RoboDK station: Deburring.rdk

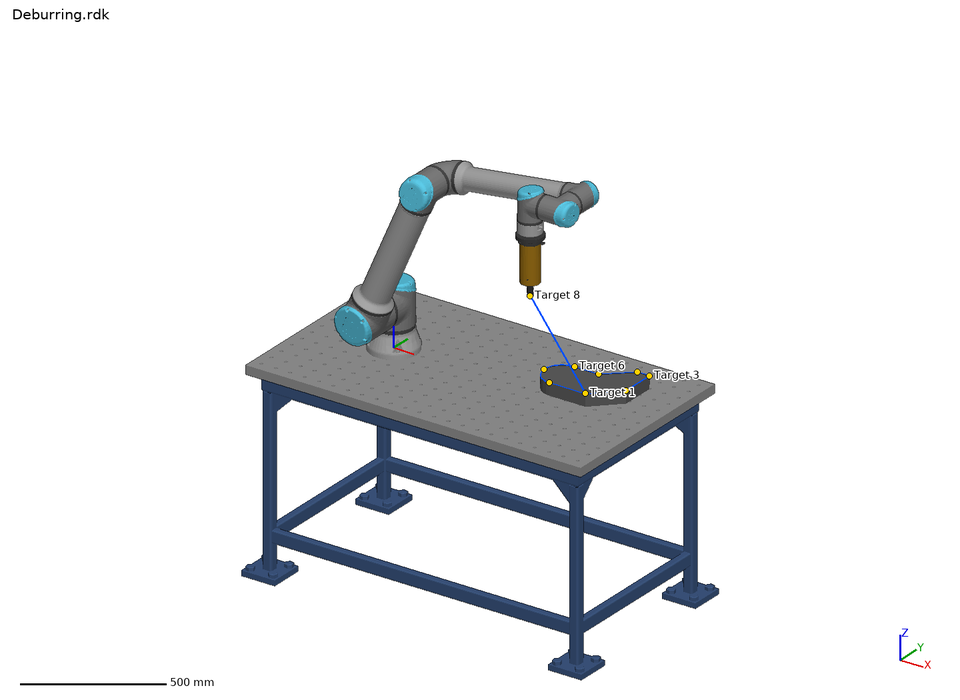
[picture v0: the station drawn from its stored meshes, robots at their saved joint values, targets as dots, program paths as lines]
Station Deburring (saved by RoboDK 5.9.2). Poses are relative to the parent item; angles as X-Y-Z fixed-axis rotations.
  - frame UR10e Base at (0, 0, 0) mm
    - robot UR10e: 6 axes, payload 10 kg, reach 1300 mm, repeatability 0.05 mm, weight 28.9 kg
        modified DH rows (alpha deg, a mm, theta deg, d mm): 0, 0, 0, 180.7; 90, 0, 180, 0; 0, 612.6, 0, 0; 0, 571.335, 0, 174.15; -90, 0, 0, 119.85; 90, 0, 180, 116.55
        joint limits [-360, -360, -360, -360, -360, -360] to [360, 360, 360, 360, 360, 360]; home [0, -90, -90, 0, 90, 0]; saved at [0, -113.502, -59.226, 82.728, 270, 180]
      - tool ATI 9150-CDB-8-11-000 Deburring Tool (Spring), TCP at (0, 0, 236.5) mm, size 103 x 103 x 235.8 mm
    - target Target 1 (Cartesian target) at (800, 0, 50) mm, rotated rx -179.28 ry 0 rz 0 deg; joints [12.276, -111.55, -108.716, -49.582, 90.702, 282.276] of UR10e
    - target Target 2 (Cartesian target) at (900, 100, 50) mm, rotated rx -179.28 ry 0 rz 0 deg; joints [17.172, -119.673, -95.84, -54.275, 90.686, 287.174] of UR10e
    - target Target 3 (Cartesian target) at (900, 240, 50) mm, rotated rx -179.28 ry 0 rz 0 deg; joints [25.472, -121.667, -92.542, -55.482, 90.648, 295.474] of UR10e
    - target Target 4 (Cartesian target) at (850, 240, 50) mm, rotated rx -179.28 ry 0 rz 0 deg; joints [26.894, -117.902, -98.773, -53.001, 90.64, 296.896] of UR10e
    - target Target 5 (Cartesian target) at (750, 150, 50) mm, rotated rx -179.28 ry 0 rz 0 deg; joints [24.18, -108.782, -112.877, -48.046, 90.655, 294.181] of UR10e
    - target Target 6 (Cartesian target) at (650, 150, 50) mm, rotated rx -179.28 ry 0 rz 0 deg; joints [27.801, -100.961, -123.659, -45.046, 90.635, 297.803] of UR10e
    - target Target 7 (Cartesian target) at (650, 0, 50) mm, rotated rx -179.28 ry 0 rz 0 deg; joints [15.174, -99.587, -125.359, -44.866, 90.693, 285.175] of UR10e
    - target Target 8 (Cartesian target) at (691.19, -174.15, 461.75) mm, rotated rx -180 ry 0 rz -90 deg; joints [0, -90, -90, -90, 90, 0] of UR10e
    - target Target 9 (Cartesian target) at (575, 75, 50) mm, rotated rx -179.28 ry 0 rz 0 deg; joints [24.517, -93.386, -132.664, -43.652, 90.653, 294.519] of UR10e
    - target Target 10 (Cartesian target) at (691.19, -174.15, 461.75) mm, rotated rx -180 ry 0 rz -90 deg; joints [0, -90, -90, -90, 90, 0] of UR10e
  - object Table 1400x800x800mm at (0, 0, 0) mm, size 1420 x 820 x 800 mm, geometry from Table.sld
  - object Random obj at (650, 0, 0) mm, size 325 x 240 x 50 mm, geometry from Random obj.step
  - program Prog1 (12 instructions, listed below)
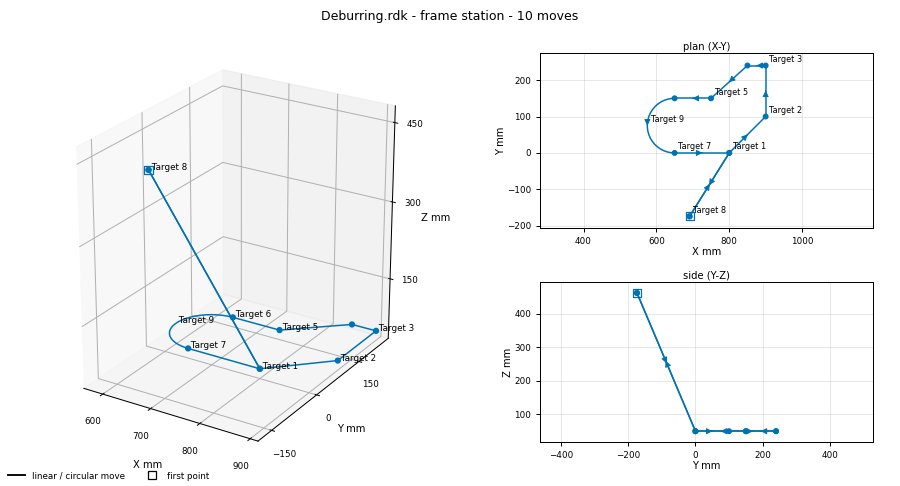
[picture p0: tool path of Deburring.rdk in frame station, 10 of 10 moves have a stored position in this frame; points joined in program order, loops and branches not executed]

--- program Prog1 (robot UR10e) ---
  Set Ref.: UR10e Base
  Set Tool: ATI 9150-CDB-8-11-000 Deburring Tool (Spring)
  MoveL (Target 8)
  MoveL (Target 1)
  MoveL (Target 2)
  MoveL (Target 3)
  MoveL (Target 4)
  MoveL (Target 5)
  MoveL (Target 6)
  MoveC (Target 9, Target 7)
  MoveL (Target 1)
  MoveL (Target 10)
